FUNCTION Init_PB_Mom_160x75 : INT

VAR_INPUT
END_VAR

VAR

END_VAR

VAR_IN_OUT
	COMP:TS_Component;
END_VAR

COMP.B_TYPE:=0;
COMP.size:=2;

END_FUNCTION

(* stored: Version 1.1.0.1, ProductVersion 3.1.4020.12
   POU Init_PB_Mom_160x75: Id {c26838f5-c21e-41d6-a420-cf8d9e7d51fb}, SpecialFunc None *)
